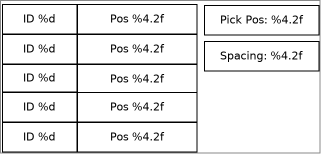
VISUALIZATION ConveyorData  // 321x154
VAR_IN_OUT
	fbConveyor : FB_Conveyor;
END_VAR
    Rectangle (77,4 120x30), "Pos %4.2f", text variable: fbConveyor.arrProductsOnConveyor[1].fPosition
    Rectangle (77,34 120x30), "Pos %4.2f", text variable: fbConveyor.arrProductsOnConveyor[2].fPosition
    Rectangle (77,64 120x30), "Pos %4.2f", text variable: fbConveyor.arrProductsOnConveyor[3].fPosition
    Rectangle (77,92 120x30), "Pos %4.2f", text variable: fbConveyor.arrProductsOnConveyor[4].fPosition
    Rectangle (77,122 120x30), "Pos %4.2f", text variable: fbConveyor.arrProductsOnConveyor[5].fPosition
    Rectangle (2,4 75x30), "ID %d", text variable: fbConveyor.arrProductsOnConveyor[1].iIDNumber
    Rectangle (2,34 75x30), "ID %d", text variable: fbConveyor.arrProductsOnConveyor[2].iIDNumber
    Rectangle (2,64 75x28), "ID %d", text variable: fbConveyor.arrProductsOnConveyor[3].iIDNumber
    Rectangle (2,92 75x30), "ID %d", text variable: fbConveyor.arrProductsOnConveyor[4].iIDNumber
    Rectangle (2,122 75x30), "ID %d", text variable: fbConveyor.arrProductsOnConveyor[5].iIDNumber
    Rectangle (204,5 115x30), "Pick Pos: %4.2f", text variable: fbConveyor.fPickLocation
    Rectangle (204,41 115x30), "Spacing: %4.2f", text variable: fbConveyor.fMinimumSpacing
END_VISUALIZATION

(* stored: Version 1.1.0.1, ProductVersion 3.1.4024.11
   Visu ConveyorData: Id {e6e094f0-5291-4413-ab72-7625c9b8364f} *)
